FUNCTION_BLOCK L3_OrderInput (* Basic Function Block Type *)
  (* Standard: 61499-2 *)
  (* Version 0.0, 2014-10-02, EQUEROL, UJI *)
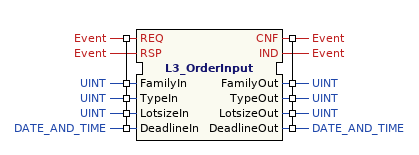
  EVENT_INPUT
    REQ WITH FamilyIn, TypeIn, LotsizeIn, DeadlineIn; (* Normal Execution Request *)
    RSP; (* Sending process completed event *)
  END_EVENT
  EVENT_OUTPUT
    CNF WITH TypeOut, LotsizeOut, DeadlineOut, FamilyOut; (* Execution Confirmation *)
    IND; (* Requested order insert completation indication *)
  END_EVENT
  VAR_INPUT
    FamilyIn : UINT; (* Part's Family *)
    TypeIn : UINT; (* Part's type *)
    LotsizeIn : UINT; (* number fo parts to be manufactured *)
    DeadlineIn : DATE_AND_TIME; (* Order's deadline *)
  END_VAR
  VAR_OUTPUT
    FamilyOut : UINT; (* Part's family *)
    TypeOut : UINT; (* Part's type *)
    LotsizeOut : UINT; (* number of parts to be manufatured *)
    DeadlineOut : DATE_AND_TIME; (* Orders's deadline *)
  END_VAR
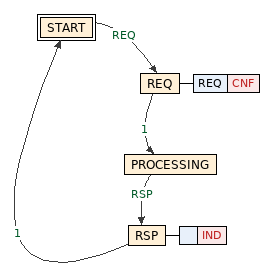
  EC_STATES
    START; (* Initial State *)
    REQ : REQ -> CNF; (* Normal execution *)
    PROCESSING;
    RSP : -> IND;
  END_STATES
  EC_TRANSITIONS
    START TO REQ := REQ;
    REQ TO PROCESSING := 1;
    PROCESSING TO RSP := RSP;
    RSP TO START := 1;
  END_TRANSITIONS
  ALGORITHM REQ IN ST: (* Normally executed algorithm *)
FamilyOut := FamilyIn;
TypeOut := TypeIn;
LotsizeOut := LotsizeIn;
DeadlineOut := DeadlineIn;
  END_ALGORITHM
END_FUNCTION_BLOCK
